TYPE Box :
STRUCT
	x				:REAL;
	y				:REAL;
	w				:REAL;
	h				:REAL;
	confidence		:REAL;
	row_index		:REAL;
	part			:REAL;
END_STRUCT
END_TYPE

(* stored: Version 1.1.0.1, ProductVersion 3.1.4024.14
   DUT Box: Id {9517058c-139b-42c3-8125-e8fc5d29678a} *)
